FUNCTION_BLOCK FB_Co2FlowModelDeviationHandler_Test EXTENDS TcUnit.FB_TestSuite
VAR_INPUT
END_VAR
VAR_OUTPUT
END_VAR
VAR
END_VAR


simpleCalculationsTest();
ifCurrentFlowIsZeroDeviationShouldBeZero();

METHOD ifCurrentFlowIsZeroDeviationShouldBeZero
VAR
	deviationHandler : FB_Co2FlowModelDeviationHandler;
END_VAR

TEST('ifCurrentFlowIsZeroDeviationShouldBeZero');

deviationHandler(
			currentFlow := 0,
			modeledFlow := 50);
					
AssertEquals_DINT(Expected := 0, Actual := deviationHandler.deviationPercentage, Message := 'Deviation not zero when current flow is zero');

TEST_FINISHED();
END_METHOD

METHOD simpleCalculationsTest
VAR
	deviationHandler : FB_Co2FlowModelDeviationHandler;
END_VAR

TEST('deviationShouldBeMinus50');

deviationHandler(
			currentFlow := 100,
			modeledFlow := 50);
					
AssertEquals_DINT(Expected := -50, Actual := deviationHandler.deviationPercentage, Message := 'Deviation not -50 when it should be');

TEST_FINISHED();

TEST('deviationShouldBePlus20');

deviationHandler(
			currentFlow := 100,
			modeledFlow := 120);
					
AssertEquals_DINT(Expected := 20, Actual := deviationHandler.deviationPercentage, Message := 'Deviation not 20 when it should be');

TEST_FINISHED();
END_METHOD

END_FUNCTION_BLOCK

(* stored: Version 1.1.0.1, ProductVersion 3.1.4024.9
   POU FB_Co2FlowModelDeviationHandler_Test: Id {dbbf9f13-0f78-4045-95eb-cf080fce2611}, SpecialFunc None
   Method ifCurrentFlowIsZeroDeviationShouldBeZero: Id {9d7019b3-e587-41fe-ac24-f8a42c05b095}
   Method simpleCalculationsTest: Id {dfe3233d-3553-4b9b-aed2-522d143efd45} *)
